FUNCTION_BLOCK FB_RS
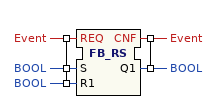
  EVENT_INPUT
    REQ WITH S, R1; (* Service Request *)
  END_EVENT
  EVENT_OUTPUT
    CNF WITH Q1; (* Confirmation of Requested Service *)
  END_EVENT
  VAR_INPUT
    S : BOOL;
    R1 : BOOL;
  END_VAR
  VAR_OUTPUT
    Q1 : BOOL;
  END_VAR
END_FUNCTION_BLOCK
